FUNCTION F_CEIL: INT;

VAR_INPUT
	iReal: REAL;

END_VAR
VAR
	tFRACResult: LREAL; //x.0000
	tReturnReal: REAL;
	
	
	tIsRemain: BOOL;
	tTRUNCResult: LREAL; //1.xxxx
	tResult: LREAL;

END_VAR

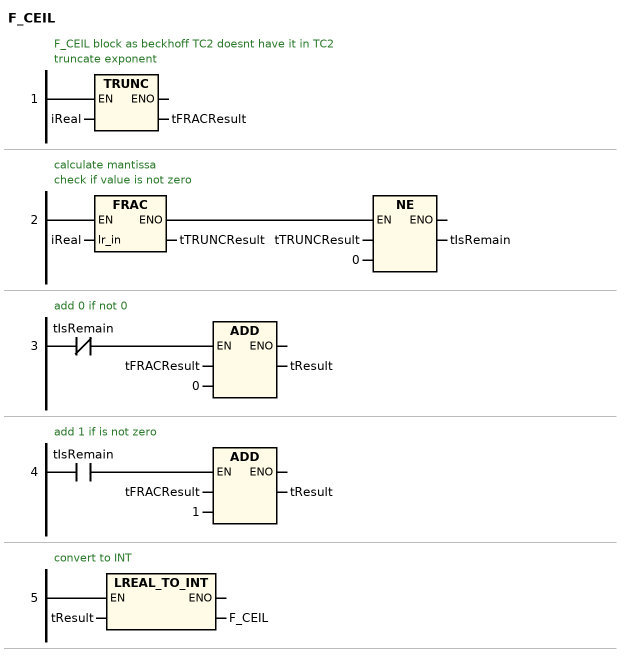
// NETWORK 1
// F_CEIL block as beckhoff TC2 doesnt have it in TC2
// truncate exponent
tFRACResult := TRUNC(iReal);

// NETWORK 2
// calculate mantissa
// check if value is not zero
tTRUNCResult := FRAC(lr_in := iReal);
tIsRemain := tTRUNCResult <> 0;

// NETWORK 3
// add 0 if not 0
IF NOT tIsRemain THEN tResult := tFRACResult + 0; END_IF

// NETWORK 4
// add 1 if is not zero
IF tIsRemain THEN tResult := tFRACResult + 1; END_IF

// NETWORK 5
// convert to INT
F_CEIL := LREAL_TO_INT(tResult);

END_FUNCTION

(* stored: Version 1.1.0.1, ProductVersion 3.1.4024.12
   POU F_CEIL: Id {b67dafea-5fa5-0c80-2d76-40da5975d8ca}, SpecialFunc None *)
